/// calibration that is determined by calibration sequences of the unit (static offsets, shifts)
TYPE ScriblyDataCalibration :
STRUCT
END_STRUCT
END_TYPE

(* stored: Version 1.1.0.1
   DUT ScriblyDataCalibration: Id {7affb8d1-ef9f-46d9-806c-7e607c048481} *)
